TYPE EL2522_Data :
STRUCT
	{attribute addProperty Name "Channel 1"}
	_1 :PTOChannel;
	{attribute addProperty Name "Channel 2"}
	_2 :PTOChannel;
END_STRUCT
END_TYPE

(* stored: Version 1.1.0.1, ProductVersion 3.1.4024.9
   DUT EL2522_Data: Id {ec39ec21-e83b-09b2-302e-2bf3831c1d7b} *)
